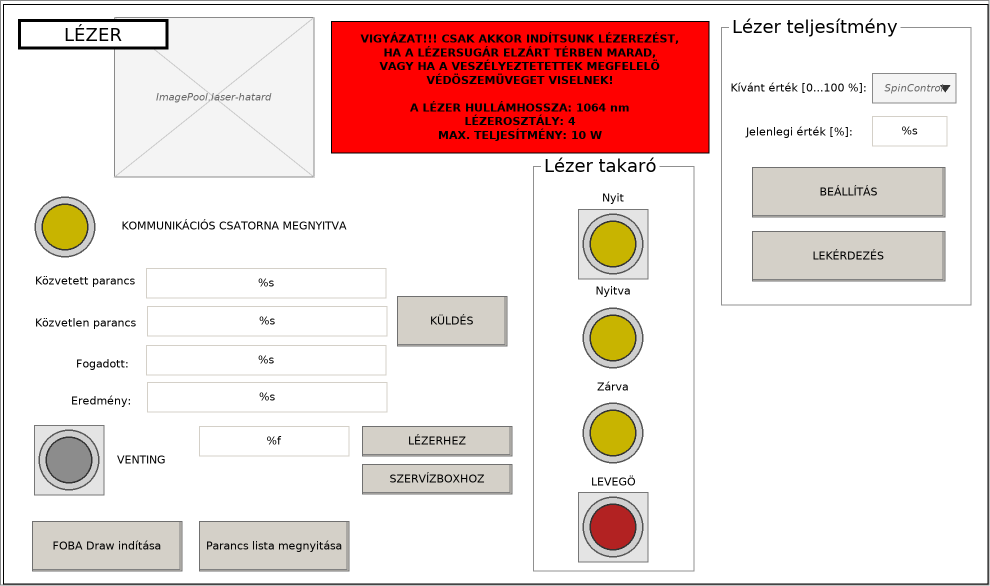
VISUALIZATION Lezer  // 990x586
    Rectangle (3,4 985x580)
    Textfield (146,268 240x30), "%s", text variable: Laser.s_InCommand
        OnMouseClick: write Laser.s_InCommand via VisuDialogs.Keypad
    Textfield (146,345 240x30), "%s", text variable: Laser.sLaserReceived
    Lamp1 (30,192 70x70), variable: GVL.bLaserCommOpen, style: Lamp-Lamp1-Yellow
    Label (106,211 256x30), "KOMMUNIKÁCIÓS CSATORNA MEGNYITVA"
    Label (70,349 65x30), "Fogadott:"
    PushSwitch (34,425 70x70), variable: AUTOMATA.bElszivasBe, behaviour: TOGGLE, style: Switch-PushSwitch-Gray
    Label (110,445 63x30), "VENTING"
    Label (24,266 114x30), "Közvetett parancs"
    Label (25,308 114x30), "Közvetlen parancs"
    Textfield (147,306 240x30), "%s", text variable: Laser.sLaserSend
        OnMouseClick: write Laser.sLaserSend via VisuDialogs.Keypad
    Button (32,521 150x50), "FOBA Draw indítása", tooltip "A jelölö lézer saját vezérlö szoftvere", pressed state: Laser.bStartFOBADraw
        OnMouseUp: execute { Laser.bStartFOBADraw:=TRUE; }
    Button (397,296 110x50), "KÜLDÉS"
        OnMouseUp: execute { Laser.iState:=1; }
    Textfield (199,426 150x30), "%f", text variable: GVL.lrVegmeroPosition
        OnMouseClick: write the text variable via VisuDialogs.Numpad, min -10000, max -1
    Image (114,17 200x160), image: ImagePool.laser-hatard
    RoundedRectangle (18,19 150x30)
    Label (18,20 150x30), "LÉZER"
    Button (199,521 150x50), "Parancs lista megnyitása", tooltip "Ultimate script-ben megírt parancsok pdf-ben", pressed state: Laser.bStartUltimate
        OnMouseUp: execute { Laser.bStartUltimate:=TRUE; }
    GroupBox (533,158 161x413), "Lézer takaró"
        PushSwitch (45,51 70x70), variable: VEGMERO.bLezertakaro, behaviour: TOGGLE, style: Switch-PushSwitch-Yellow
        Label (55,30 50x20), "Nyit"
        Lamp1 (45,145 70x70), variable: VEGMERO.bLezertakaroNyitva, style: Lamp-Lamp1-Yellow
        Label (55,123 50x20), "Nyitva"
        Lamp1 (45,240 70x70), variable: VEGMERO.bLezertakaroZarva, style: Lamp-Lamp1-Yellow
        Label (55,219 50x20), "Zárva"
        Group (45,309 70x95)
            PushSwitch (0,25 70x70), variable: MAIN.bLevego, behaviour: TOGGLE, style: Switch-PushSwitch-Red
            Label (1,0 69x30), "LEVEGÖ"
    RoundedRectangle (331,21 378x132), "VIGYÁZAT!!! CSAK AKKOR INDÍTSUNK LÉZEREZÉST, HA A LÉZERSUGÁR ELZÁRT TÉRBEN MARAD, VAGY HA A VESZÉLYEZTETETTEK MEGFELELÖ VÉDÖSZEMÜVEGET VISELNEK! A LÉZER HULLÁMHOSSZA: 1064 nm LÉZEROSZTÁLY: 4 MAX. TELJESÍTMÉNY: 10 W"
    Button (362,426 150x30), "LÉZERHEZ"
        OnMouseUp: execute { PISTITENGELY.lrPistiPosition:=GVL.lrVegmeroPosition; PISTITENGELY.sPistiAxisCommand:='MOVE'; }
    Button (362,464 150x30), "SZERVÍZBOXHOZ"
        OnMouseUp: execute { PISTITENGELY.lrPistiPosition:=GVL.lrPtSzervizbox; PISTITENGELY.sPistiAxisCommand:='MOVE'; }
    Textfield (147,382 240x30), "%s", text variable: Laser.sLaserReceived
    Label (66,386 70x30), "Eredmény:"
    GroupBox (721,19 250x286), "Lézer teljesítmény"
        SpinControl (151,54 84x30), variable: Laser.iWishPower
            OnMouseClick: write Laser.iWishPower via VisuDialogs.Numpad, min 0, max 100
        Label (11,54 133x30), "Kívánt érték [0...100 %]:"
        Label (12,98 133x30), "Jelenlegi érték [%]:"
        Textfield (151,97 75x30), "%s", text variable: Laser.iSetPower
        Button (31,148 193x50), "BEÁLLÍTÁS"
            OnMouseUp: execute {
                Laser.sLaserSend:=CONCAT('SetIntensity;',
                				  CONCAT(INT_TO_STRING(Laser.iWishPower),';'));
                Laser.iState:=1;
            }
        Button (31,212 193x50), "LEKÉRDEZÉS"
            OnMouseUp: execute { Laser.sLaserSend:='GetIntensity;'; Laser.iState:=1; }
END_VISUALIZATION

(* stored: Version 1.1.0.1, ProductVersion 3.1.4024.11
   Visu Lezer: Id {ca7a39f1-1dd7-4f2a-b538-c4c998af8abd} *)
